FUNCTION Buffer_Layout_Set_UDInt_Array : UINT
VAR_INPUT
END_VAR
VAR
END_VAR

END_FUNCTION

(* stored: Version 1.1.0.1, ProductVersion 3.1.4024.10
   POU Buffer_Layout_Set_UDInt_Array: Id {4da5b8ee-4a07-412a-b657-ec8182f244ae}, SpecialFunc None *)
